PROGRAM MASTER2_IO_Map
VAR
	BYTE_AS_BIT_0: BYTE_AS_BIT;
	BYTE_AS_BIT_1: BYTE_AS_BIT;
	BYTE_AS_BIT_2: BYTE_AS_BIT;
	BYTE_AS_BIT_3: BYTE_AS_BIT;

	BIT_AS_BYTE_0: BIT_AS_BYTE;
	BIT_AS_BYTE_1: BIT_AS_BYTE;
	BIT_AS_BYTE_2: BIT_AS_BYTE;
	BIT_AS_BYTE_3: BIT_AS_BYTE;
	
	OP10_MAS2_PORT1_BYTE1_DI_MODULE_1 AT %I* : BYTE;
	OP10_MAS2_PORT1_BYTE2_DI_MODULE_1 AT %I* : BYTE;
	OP10_MAS2_PORT2_BYTE1_DI_MODULE_2 AT %I* : BYTE;
	OP10_MAS2_PORT2_BYTE2_DI_MODULE_2 AT %I* : BYTE;	

	
END_VAR

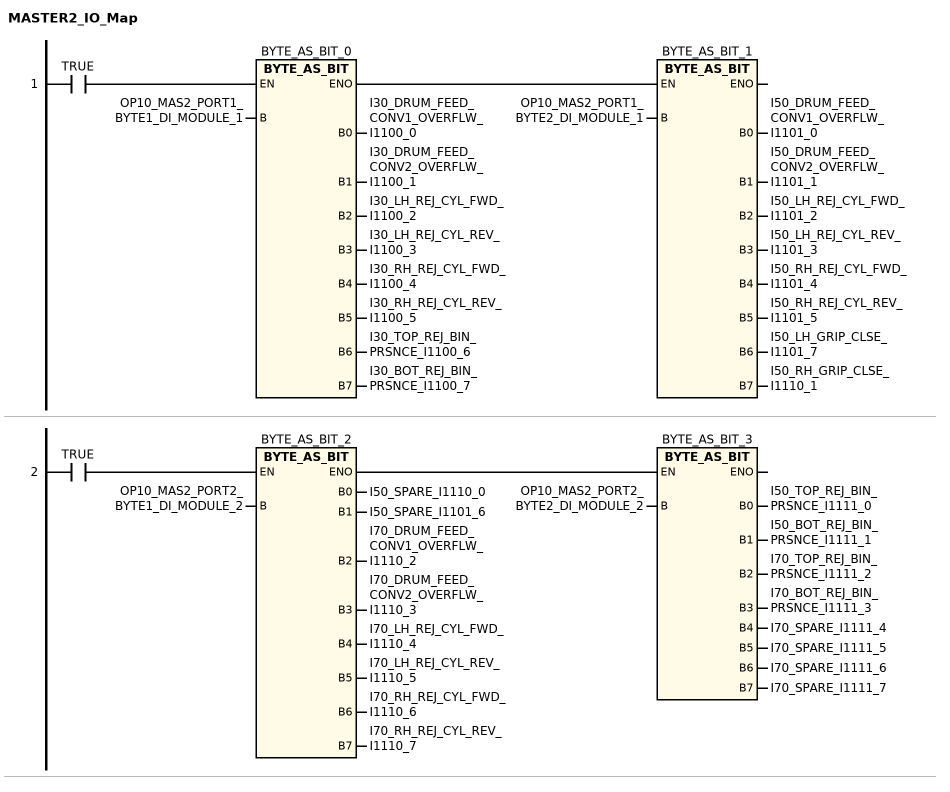
// NETWORK 1
BYTE_AS_BIT_0(
    B := OP10_MAS2_PORT1_BYTE1_DI_MODULE_1,
    B0 => I30_DRUM_FEED_CONV1_OVERFLW_I1100_0,
    B1 => I30_DRUM_FEED_CONV2_OVERFLW_I1100_1,
    B2 => I30_LH_REJ_CYL_FWD_I1100_2,
    B3 => I30_LH_REJ_CYL_REV_I1100_3,
    B4 => I30_RH_REJ_CYL_FWD_I1100_4,
    B5 => I30_RH_REJ_CYL_REV_I1100_5,
    B6 => I30_TOP_REJ_BIN_PRSNCE_I1100_6,
    B7 => I30_BOT_REJ_BIN_PRSNCE_I1100_7); // BYTE_AS_BIT
BYTE_AS_BIT_1(
    B := OP10_MAS2_PORT1_BYTE2_DI_MODULE_1,
    B0 => I50_DRUM_FEED_CONV1_OVERFLW_I1101_0,
    B1 => I50_DRUM_FEED_CONV2_OVERFLW_I1101_1,
    B2 => I50_LH_REJ_CYL_FWD_I1101_2,
    B3 => I50_LH_REJ_CYL_REV_I1101_3,
    B4 => I50_RH_REJ_CYL_FWD_I1101_4,
    B5 => I50_RH_REJ_CYL_REV_I1101_5,
    B6 => I50_LH_GRIP_CLSE_I1101_7,
    B7 => I50_RH_GRIP_CLSE_I1110_1); // BYTE_AS_BIT

// NETWORK 2
BYTE_AS_BIT_2(
    B := OP10_MAS2_PORT2_BYTE1_DI_MODULE_2,
    B0 => I50_SPARE_I1110_0,
    B1 => I50_SPARE_I1101_6,
    B2 => I70_DRUM_FEED_CONV1_OVERFLW_I1110_2,
    B3 => I70_DRUM_FEED_CONV2_OVERFLW_I1110_3,
    B4 => I70_LH_REJ_CYL_FWD_I1110_4,
    B5 => I70_LH_REJ_CYL_REV_I1110_5,
    B6 => I70_RH_REJ_CYL_FWD_I1110_6,
    B7 => I70_RH_REJ_CYL_REV_I1110_7); // BYTE_AS_BIT
BYTE_AS_BIT_3(
    B := OP10_MAS2_PORT2_BYTE2_DI_MODULE_2,
    B0 => I50_TOP_REJ_BIN_PRSNCE_I1111_0,
    B1 => I50_BOT_REJ_BIN_PRSNCE_I1111_1,
    B2 => I70_TOP_REJ_BIN_PRSNCE_I1111_2,
    B3 => I70_BOT_REJ_BIN_PRSNCE_I1111_3,
    B4 => I70_SPARE_I1111_4,
    B5 => I70_SPARE_I1111_5,
    B6 => I70_SPARE_I1111_6,
    B7 => I70_SPARE_I1111_7); // BYTE_AS_BIT

END_PROGRAM

(* stored: Version 1.1.0.1, ProductVersion 3.1.4024.11
   POU MASTER2_IO_Map: Id {7f66d372-364b-4c22-80c0-c6bc97964263}, SpecialFunc None *)
